FUNCTION_BLOCK FB_Stan_Suspending EXTENDS FB_SITP_Element
VAR

END_VAR

METHOD FB_init : BOOL
VAR_INPUT
	bInitRetains : BOOL; // if TRUE, the retain variables are initialized (warm start / cold start)
	bInCopyCode : BOOL;  // if TRUE, the instance afterwards gets moved into the copy code (online change)
END_VAR
THIS^.PrzypiszTekstDo (refstEtykieta := THIS^.stNazwa, eJezyk := B_Baza.E_Jezyki.pl, wsTekst	:= "Zawieszanie");
THIS^.PrzypiszTekstDo (refstEtykieta := THIS^.stNazwa, eJezyk := B_Baza.E_Jezyki.de, wsTekst	:= "Aussetzen");  
THIS^.PrzypiszTekstDo (refstEtykieta := THIS^.stNazwa, eJezyk := B_Baza.E_Jezyki.en, wsTekst	:= "Suspending");
END_METHOD

METHOD PUBLIC WywolajAkcjePBDlaStanu : BOOL
VAR_INPUT
	iNumerPB				: INT;
END_VAR
WywolajAkcjePBDlaStanu			:= THIS^.refstDaneSITP.refarrPB [iNumerPB].SP_Suspending ();
END_METHOD

(*			
	EVERDE sp. z o.o.
	Rafał Osajda		18.06.2025		TC 4024.66
	Zwraca true jak wyjście ze stanu jest możliwe
*)
METHOD PUBLIC ZwrocCzyMoznaWyjscZeStanu : BOOL
//warunki wyjść dla każdego ze stanów osobnym FB
IF (THIS^.refstDaneSITP.ePolecenieZmianyStanu = E_SITP_PolecenieZmianyStanu.Abort) THEN
	IF (THIS^.refstDaneSITP.arrStanyWlaczoneWTrybie [B_Baza.E_StanyPracy.Aborting]) THEN
		ZwrocCzyMoznaWyjscZeStanu					:= THIS^.ZgodaNaZmianeStanu (B_Baza.E_StanyPracy.Aborting);
	ELSE
		ZwrocCzyMoznaWyjscZeStanu					:= THIS^.BrakZgodyNaZmieneStanu (2);	//Stan do którego chcemy przejść jest wylaczony
	END_IF
ELSIF (THIS^.refstDaneSITP.ePolecenieZmianyStanu = E_SITP_PolecenieZmianyStanu.Stop) THEN
	IF (THIS^.refstDaneSITP.arrStanyWlaczoneWTrybie [B_Baza.E_StanyPracy.Stopping]) THEN
		ZwrocCzyMoznaWyjscZeStanu					:= THIS^.ZgodaNaZmianeStanu (B_Baza.E_StanyPracy.Stopping);
	ELSE
		ZwrocCzyMoznaWyjscZeStanu					:= THIS^.BrakZgodyNaZmieneStanu (2);	//Stan do którego chcemy przejść jest wylaczony
	END_IF
ELSIF (THIS^.refstDaneSITP.ePolecenieZmianyStanu <> E_SITP_PolecenieZmianyStanu.Abort AND
		THIS^.refstDaneSITP.ePolecenieZmianyStanu <> E_SITP_PolecenieZmianyStanu.Stop AND 
		THIS^.refstDaneSITP.ePolecenieZmianyStanu <> E_SITP_PolecenieZmianyStanu.brak) THEN
	ZwrocCzyMoznaWyjscZeStanu						:= THIS^.BrakZgodyNaZmieneStanu (1);	//Bledny rozkaz dla zmiany stanu
ELSIF (THIS^.refstDaneSITP.refbWyjdzZestanuAktywnego) THEN
	IF (THIS^.refstDaneSITP.arrStanyWlaczoneWTrybie [B_Baza.E_StanyPracy.Suspended]) THEN
		ZwrocCzyMoznaWyjscZeStanu					:= THIS^.ZgodaNaZmianeStanu (B_Baza.E_StanyPracy.Suspended);
	ELSE
		ZwrocCzyMoznaWyjscZeStanu					:= THIS^.BrakZgodyNaZmieneStanu (2);	//Stan do którego chcemy przejść jest wylaczony
	END_IF
ELSE
	ZwrocCzyMoznaWyjscZeStanu						:= THIS^.BrakZgodyNaZmieneStanu (3);	//Brak polecenia wyjsciua z stanu aktywnego - ing
END_IF
END_METHOD

END_FUNCTION_BLOCK

(* stored: Version 1.1.0.1
   POU FB_Stan_Suspending: Id {f00f0fb7-b820-05bd-1895-51e771c5dafd}, SpecialFunc None
   Method FB_init: Id {7b07cbaa-a3f8-052f-2048-8021c9c591e7}
   Method WywolajAkcjePBDlaStanu: Id {b2248962-94fd-07fa-0541-674b75b4e74e}
   Method ZwrocCzyMoznaWyjscZeStanu: Id {ad139067-1427-02f5-28bf-5d65f4e90b96} *)
